ABB RobotStudio station: Solution_1.rspag

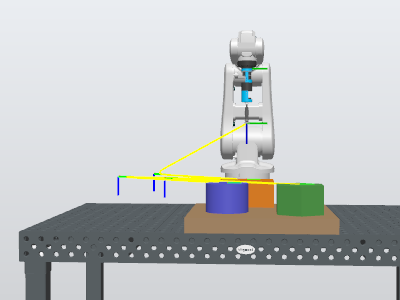
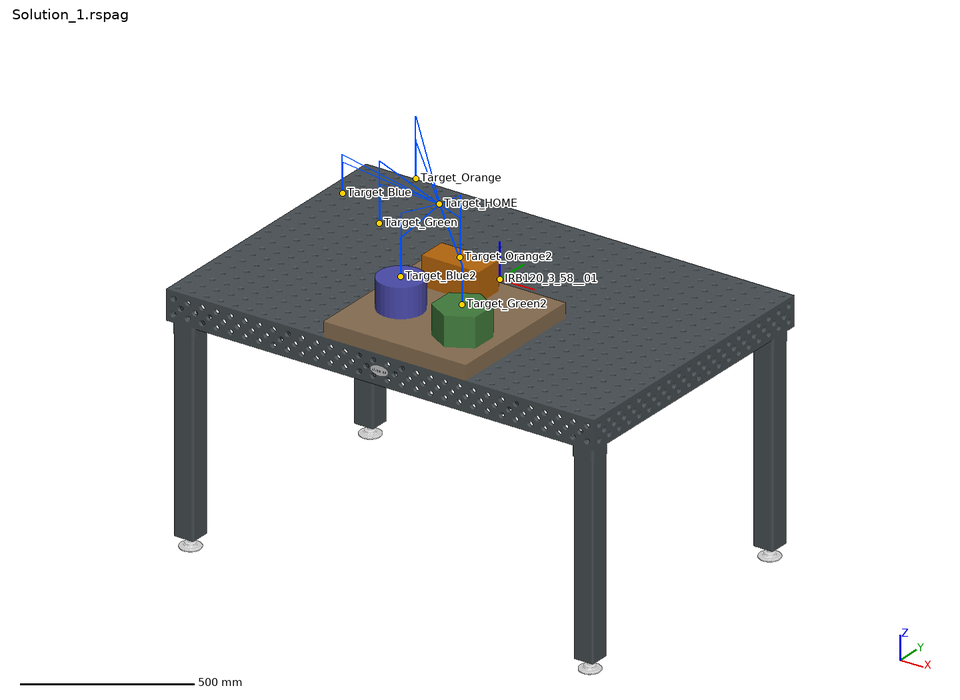
[picture v1: parts stored in the station drawn from their meshes, with robot base, taught points and paths (robot models come from the ABB library and are not in the file)]
--- station ---
Station Solution_1_Tutorial (saved by RobotStudio 22.3.10190.2)
Controller Controller1, task T_ROB1: task frame (RAPID world) sits at (0, 100, 830) mm, rotated rx 0 ry 0 rz -90 deg in the station
Controller Controller1
  mechanical unit ROB_1: IRB120_3_58__01, 6 joints, base frame (0, 0, 0) mm
Layout (positions relative to the parent item):
  - table [part] at (-200, -500, 830) mm, size 500 x 500 x 50 mm
  - object_1 [part] at (-200, -500, 830) mm, size 200 x 100 x 150 mm
  - object_2 [part] at (-200, -500, 830) mm, size 149.5 x 149.7 x 150 mm
  - object_3 [part] at (-200, -500, 830) mm, size 155.5 x 179.5 x 150 mm
  - siegmund_1500_1000 [part], size 1500 x 1010.3 x 830 mm
  - object_11 [part] at (-200, -500, 830) mm, size 200 x 100 x 150 mm
  - object_22 [part] at (-200, -500, 830) mm, size 149.5 x 149.7 x 150 mm
  - object_33 [part] at (-200, -500, 830) mm, size 155.5 x 179.5 x 150 mm
  - IRB120_3_58__01 [mechanism, from Robots\IRB120_3_58_G_01.rslib] at (0, 100, 830) mm, rotated rx 0 ry 0 rz -90 deg; joint values [0, 0, 0, 0, 1.5708, 0] (rad or m)
  - smc_gripper [mechanism, from Gripper_RS_tool\smc_gripper.rslib] at (0, -202, 1388) mm, rotated rx 180 ry 0 rz 90 deg
  - Positioner [smart component, from Components\Positioner.rslib]
      properties: Object=object_1; Position=[-0.6 -0.15 0.83]; Orientation=[0 0 0]; Reference=Global; ReferenceObject=(none)
  - Positioner_2 [smart component, from Components\Positioner.rslib]
      properties: Object=object_2; Position=[-0.65 -0.15 0.83]; Orientation=[0 0 0]; Reference=Global; ReferenceObject=(none)
  - Positioner_3 [smart component, from Components\Positioner.rslib]
      properties: Object=object_3; Position=[-0.7 -0.2 0.83]; Orientation=[0 0 0]; Reference=Global; ReferenceObject=(none)
  - Attacher [smart component, from Components\Attacher.rslib]
      properties: Parent=smc_gripper; Flange=0; Child=object_1; Mount=false; Offset=[0 0 0]; Orientation=[0 0 0]
  - Attacher_2 [smart component, from Components\Attacher.rslib]
      properties: Parent=smc_gripper; Flange=0; Child=object_2; Mount=false; Offset=[0 0 0]; Orientation=[0 0 0]
  - Attacher_3 [smart component, from Components\Attacher.rslib]
      properties: Parent=smc_gripper; Flange=0; Child=object_3; Mount=false; Offset=[0 0 0]; Orientation=[0 0 0]
  - Detacher [smart component, from Components\Detacher.rslib]
      properties: Child=object_1; KeepPosition=true
  - Detacher_2 [smart component, from Components\Detacher.rslib]
      properties: Child=object_2; KeepPosition=true
  - Detacher_3 [smart component, from Components\Detacher.rslib]
      properties: Child=object_3; KeepPosition=true
Attachment: smc_gripper is attached to IRB120_3_58__01 / Link6
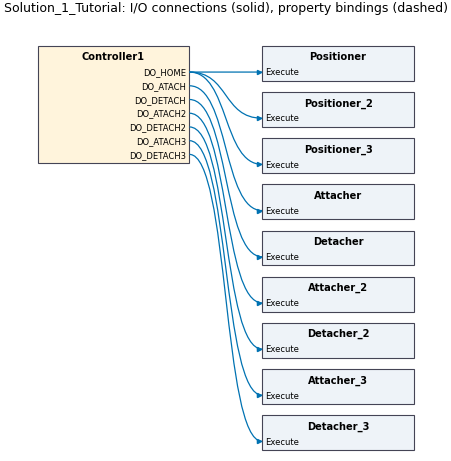
Station logic (signal -> signal, property => property):
  Controller1.DO_HOME -> Positioner.Execute
  Controller1.DO_HOME -> Positioner_2.Execute
  Controller1.DO_HOME -> Positioner_3.Execute
  Controller1.DO_ATACH -> Attacher.Execute
  Controller1.DO_DETACH -> Detacher.Execute
  Controller1.DO_ATACH2 -> Attacher_2.Execute
  Controller1.DO_DETACH2 -> Detacher_2.Execute
  Controller1.DO_ATACH3 -> Attacher_3.Execute
  Controller1.DO_DETACH3 -> Detacher_3.Execute
Targets, tools, work objects and paths stored in the station and not in the controller backup, written as RAPID:
! task T_ROB1
MODULE Module1
  PROC Path_10()
    MoveL Target_HOME,v1000,z100,smc_gripper\WObj:=wobj0;
    MoveL Target_Orange,v1000,z100,smc_gripper\WObj:=wobj0;
    MoveL Target_Orange2,v1000,z100,smc_gripper\WObj:=wobj0;
    MoveL Target_Blue,v1000,z100,smc_gripper\WObj:=wobj0;
    MoveL Target_Blue2,v1000,z100,smc_gripper\WObj:=wobj0;
    MoveL Target_Green,v1000,z100,smc_gripper\WObj:=wobj0;
    MoveL Target_Green2,v1000,z100,smc_gripper\WObj:=wobj0;
  ENDPROC
ENDMODULE


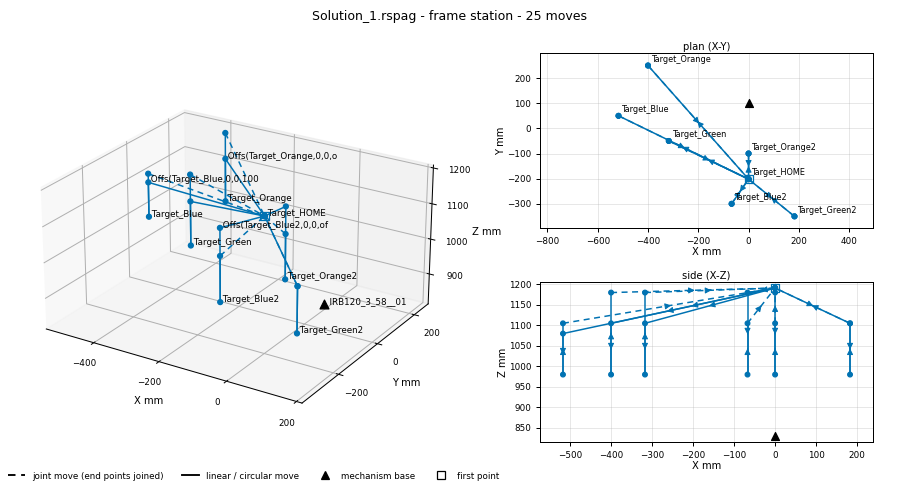
[picture p0: tool path of Solution_1.rspag in frame station, 25 of 25 moves have a stored position in this frame; points joined in program order, loops and branches not executed]
--- Backups/Controller1/RAPID/TASK1/PROGMOD/CalibData.mod ---
MODULE CalibData
    PERS tooldata smc_gripper:=[TRUE,[[0,0.004,197.001],[1,0,0,0]],[1,[0.207,-0.496,71.18],[1,0,0,0],0,0,0]];
ENDMODULE

--- Backups/Controller1/RAPID/TASK1/PROGMOD/Module1.mod ---
MODULE Module1
    CONST robtarget Target_HOME:=[[302,0.004,360.999],[0,0,1,0],[0,0,0,0],[9E+09,9E+09,9E+09,9E+09,9E+09,9E+09]];
    CONST robtarget Target_Orange:=[[-150,-400,150],[0,0,1,0],[0,0,0,0],[9E+09,9E+09,9E+09,9E+09,9E+09,9E+09]];
    CONST robtarget Target_Orange2:=[[200,0,150],[0,0,1,0],[0,0,0,0],[9E+09,9E+09,9E+09,9E+09,9E+09,9E+09]];
    CONST robtarget Target_Blue:=[[50,-517.298,150],[0,0,1,0],[0,0,0,0],[9E+09,9E+09,9E+09,9E+09,9E+09,9E+09]];
    CONST robtarget Target_Blue2:=[[400,-67.298,150],[0,0,1,0],[0,0,0,0],[9E+09,9E+09,9E+09,9E+09,9E+09,9E+09]];
    CONST robtarget Target_Green:=[[150,-317.298,150],[0,0,1,0],[0,0,0,0],[9E+09,9E+09,9E+09,9E+09,9E+09,9E+09]];
    CONST robtarget Target_Green2:=[[450,182.702,150],[0,0,1,0],[0,0,0,0],[9E+09,9E+09,9E+09,9E+09,9E+09,9E+09]];
    VAR num offset_z:=200;
    VAR num offset_zn:=125;


    PROC main()
        !SETUP
        PulseDO DO_DETACH;
        PulseDO DO_DETACH2;
        PulseDO DO_DETACH3;
        PulseDO DO_HOME;
        MoveJ Target_HOME,v100,fine,smc_gripper;
        !ORANGE
        MoveL Offs(Target_Orange,0,0,offset_zn),v100,z50,smc_gripper;
        MoveL Target_Orange,v100,fine,smc_gripper;
        PulseDO DO_ATACH;
        WaitTime 0.5;
        MoveL Offs(Target_Orange,0,0,offset_z),v100,z50,smc_gripper;
        MoveJ Target_HOME,v100,z50,smc_gripper;
        MoveL Offs(Target_Orange2,0,0,offset_z),v100,z50,smc_gripper;
        MoveL Target_Orange2,v100,fine,smc_gripper;
        PulseDO DO_DETACH;
        WaitTime 0.5;
        MoveL Offs(Target_Orange2,0,0,offset_zn),v100,z50,smc_gripper;
        MoveJ Target_HOME,v100,fine,smc_gripper;
        !BLUE
        MoveL Offs(Target_Blue,0,0,100),v100,z50,smc_gripper;
        MoveL Target_Blue,v100,fine,smc_gripper;
        PulseDO DO_ATACH2;
        WaitTime 0.5;
        MoveL Offs(Target_Blue,0,0,offset_zn),v100,z50,smc_gripper;
        MoveJ Target_HOME,v100,z50,smc_gripper;
        MoveL Offs(Target_Blue2,0,0,offset_z),v100,z50,smc_gripper;
        MoveL Target_Blue2,v100,fine,smc_gripper;
        PulseDO DO_DETACH2;
        WaitTime 0.5;
        MoveL Offs(Target_Blue2,0,0,offset_zn),v100,z50,smc_gripper;
        MoveJ Target_HOME,v100,fine,smc_gripper;
        !GREEN
        MoveL Offs(Target_Green,0,0,offset_zn),v100,z50,smc_gripper;
        MoveL Target_Green,v100,fine,smc_gripper;
        PulseDO DO_ATACH3;
        WaitTime 0.5;
        MoveL Offs(Target_Green,0,0,offset_z),v100,z50,smc_gripper;
        MoveJ Target_HOME,v100,z50,smc_gripper;
        MoveL Offs(Target_Green2,0,0,offset_zn),v100,z50,smc_gripper;
        MoveL Target_Green2,v100,fine,smc_gripper;
        PulseDO DO_DETACH3;
        WaitTime 0.5;
        MoveL Offs(Target_Green2,0,0,offset_zn),v100,z50,smc_gripper;
        MoveJ Target_HOME,v100,fine,smc_gripper;
    ENDPROC
ENDMODULE

--- Backups/Controller1/SYSPAR/EIO.cfg ---
EIO:CFG_1.0:6:1::
#
EIO_SIGNAL:

      -Name "DO_HOME" -SignalType "DO"

      -Name "DO_ATACH" -SignalType "DO"

      -Name "DO_ATACH2" -SignalType "DO"

      -Name "DO_ATACH3" -SignalType "DO"

      -Name "DO_DETACH" -SignalType "DO"

      -Name "DO_DETACH2" -SignalType "DO"

      -Name "DO_DETACH3" -SignalType "DO"
